// TwinCAT 3 PLC project PLC
// ProgramVersion: 3.1.4023.0
// libraries:
//   Tc2_Standard, * (Beckhoff Automation GmbH)
//   Tc2_System, * (Beckhoff Automation GmbH)
//   Tc3_Module, * (Beckhoff Automation GmbH)
// project tree:
//   / PlcTask.TcTTO (not stored)
//   POUs/ MAIN.TcPOU, Sum.TcPOU

// ---- POUs/MAIN.TcPOU
PROGRAM MAIN
VAR
END_VAR

Sum(3.4, 5.1);

END_PROGRAM

// ---- POUs/Sum.TcPOU
FUNCTION Sum : LREAL
VAR_INPUT
    var1 : LREAL;
    var2 : LREAL;
END_VAR
VAR
    total : LREAL;
END_VAR

// Body

END_FUNCTION
